TYPE "PLCtoMES_PrintExchange_ext"
VERSION : 0.1
   STRUCT
      Load_PrintReq : Bool;
      Load_DataMatrixCheckReq : Bool;
      Load_Spare : Bool;
      Load_Spare_1 : Bool;
      Load_Spare_2 : Bool;
      Load_Spare_3 : Bool;
      Load_Spare_4 : Bool;
      Load_Spare_5 : Bool;
      Spare : Byte;
   END_STRUCT;

END_TYPE

